FUNCTION_BLOCK FB_LPhotonEnergy
VAR_INPUT
END_VAR
VAR_OUTPUT
END_VAR
VAR_IN_OUT
	BP : ST_BeamParams;
END_VAR
VAR
	{attribute 'pytmc' := '
        pv: eEnrg
        link: BEND:DMPH:400:BACT
        field: EGU GeV
    '}
    fbHgvpuElectronEnergy : FB_LREALFromEPICS;
	
    {attribute 'pytmc' := '
        pv: EEnergy
		io: i
        field: DESC Electron Energy
        field: EGU GeV
    '}
    fElectronEnergyVal : LREAL;
    
    {attribute 'pytmc' := '
        pv: EEnergyValid
		io: i
        field: DESC Electron Energy Valid
    '}
    bElectronEnergyValid : BOOL;
    
	{attribute 'pytmc' := '
        pv: UND
        link: USEG:UNDH:
    '}
    fbHgvpu : FB_Hgvpu;
	
	nCurrentPhotonEnergyBitmask : UINT;
	nTargetPhotonEnergyBitmask : UINT;
END_VAR

// Update PVs
fbHgvpuElectronEnergy();

fbHgvpu(fbElectronEnergy:=fbHgvpuElectronEnergy);

//Update BP
nCurrentPhotonEnergyBitmask := F_eVRangeCalculator(fbHgvpu.fCurrentPhotonEnergy, nCurrentPhotonEnergyBitmask);
nTargetPhotonEnergyBitmask := F_eVRangeCalculator(fbHgvpu.fTargetPhotonEnergy, nTargetPhotonEnergyBitmask);

BP.neVRange := nCurrentPhotonEnergyBitmask OR nTargetPhotonEnergyBitmask;

END_FUNCTION_BLOCK

(* stored: Version 1.1.0.1, ProductVersion 3.1.4022.18
   POU FB_LPhotonEnergy: Id {bdcefa0d-d4a1-4d69-beca-093e09b6a2b2}, SpecialFunc None *)
